{attribute addProperty BoxType "KL9900-0056"}
{attribute addProperty Id "Key_1AT %I*BOOL000Key_2AT %I*BOOL000Key_3AT %I*BOOL000Key_4AT %I*BOOL000Key_5AT %I*BOOL000Key_6AT %I*BOOL000Key_7AT %I*BOOL000Key_8AT %I*BOOL000Key_9AT %I*BOOL000Key_10AT %I*BOOL000Key_11AT %I*BOOL000Key_12AT %I*BOOL000LED_1AT %Q*BOOL000LED_2AT %Q*BOOL000LED_3AT %Q*BOOL000LED_4AT %Q*BOOL000LED_5AT %Q*BOOL000LED_6AT %Q*BOOL000LED_7AT %Q*BOOL000LED_8AT %Q*BOOL000LED_9AT %Q*BOOL000LED_10AT %Q*BOOL000LED_11AT %Q*BOOL000LED_12AT %Q*BOOL000"}
{attribute addProperty CRC "312211932"}
{attribute addProperty SizeInBites "0"}
{attribute addProperty SizeInBytes "0"}
TYPE Channel_129BF9DC :
STRUCT
	{attribute addProperty Name "Key_1"}
	Key_1 AT %I* : BOOL;
	{attribute addProperty Name "Key_2"}
	Key_2 AT %I* : BOOL;
	{attribute addProperty Name "Key_3"}
	Key_3 AT %I* : BOOL;
	{attribute addProperty Name "Key_4"}
	Key_4 AT %I* : BOOL;
	{attribute addProperty Name "Key_5"}
	Key_5 AT %I* : BOOL;
	{attribute addProperty Name "Key_6"}
	Key_6 AT %I* : BOOL;
	{attribute addProperty Name "Key_7"}
	Key_7 AT %I* : BOOL;
	{attribute addProperty Name "Key_8"}
	Key_8 AT %I* : BOOL;
	{attribute addProperty Name "Key_9"}
	Key_9 AT %I* : BOOL;
	{attribute addProperty Name "Key_10"}
	Key_10 AT %I* : BOOL;
	{attribute addProperty Name "Key_11"}
	Key_11 AT %I* : BOOL;
	{attribute addProperty Name "Key_12"}
	Key_12 AT %I* : BOOL;
	{attribute addProperty Name "LED_1"}
	LED_1 AT %Q* : BOOL;
	{attribute addProperty Name "LED_2"}
	LED_2 AT %Q* : BOOL;
	{attribute addProperty Name "LED_3"}
	LED_3 AT %Q* : BOOL;
	{attribute addProperty Name "LED_4"}
	LED_4 AT %Q* : BOOL;
	{attribute addProperty Name "LED_5"}
	LED_5 AT %Q* : BOOL;
	{attribute addProperty Name "LED_6"}
	LED_6 AT %Q* : BOOL;
	{attribute addProperty Name "LED_7"}
	LED_7 AT %Q* : BOOL;
	{attribute addProperty Name "LED_8"}
	LED_8 AT %Q* : BOOL;
	{attribute addProperty Name "LED_9"}
	LED_9 AT %Q* : BOOL;
	{attribute addProperty Name "LED_10"}
	LED_10 AT %Q* : BOOL;
	{attribute addProperty Name "LED_11"}
	LED_11 AT %Q* : BOOL;
	{attribute addProperty Name "LED_12"}
	LED_12 AT %Q* : BOOL;
END_STRUCT
END_TYPE

(* stored: Version 1.2.0.0, ProductVersion 3.1.4024.9
   DUT Channel_129BF9DC: Id {a7fad01a-91ee-4058-98f9-d207edb3dc0f} *)
